Universal Robots PolyScope program: MarinaFerranP3.urp

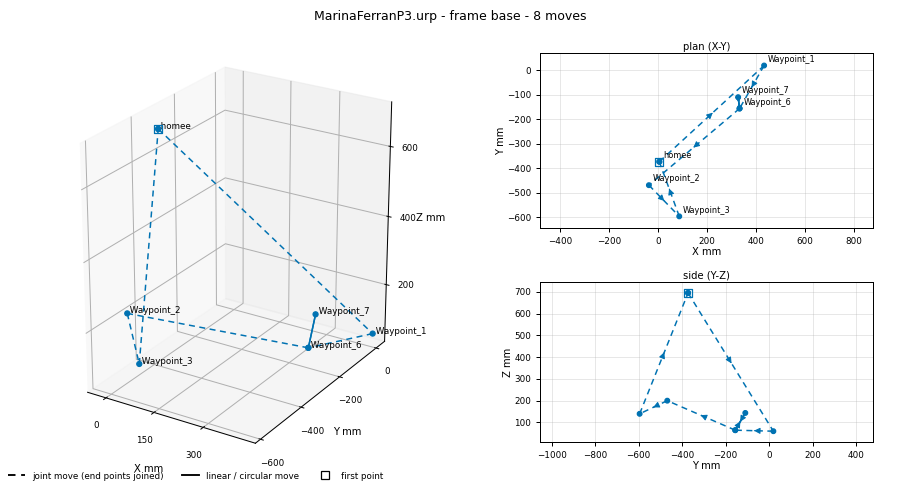
[picture p0: tool path of MarinaFerranP3.urp in frame base, 8 of 8 moves have a stored position in this frame; points joined in program order, loops and branches not executed]
Program MarinaFerranP3 (installation=default directory=/programs createdIn=5.14.5 lastSavedIn=5.14.5 robotSerialNumber=20195300809)
Calibrated DH parameters: a=[-0.000085, -0.20076, -0.212369, 0.000121, -0.000118, 0]; d=[0.15185, -26.306375, 24.753047, 1.684739, 0.085386, 0.092088]; alpha=[1.572149, -0.00522, -0.011864, 1.571339, -1.571085, 0]; deltaTheta=[0, 0.599885, -0.513355, -0.086555, 0.000006, 0]
InitVariablesNode
Robot Program (runOnlyOnce=false)
  URCap Gripper (Robotiq_Grippers, Robotiq Inc.) dataModel(position=0.0, force=100.0, speed=100.0, positionInDouble=0.0, forceInDouble=100.0, speedInDouble=100.0, slaveIds=[9], blocking=true)
  MoveJ speed 60 deg/s, acceleration 80 deg/s^2 (useActiveTCP=true) feature=Base
    Waypoint homee: TCP in base x=5.952 y=-372.701 z=694.671 mm, rx=-0.0179 ry=2.2102 rz=-2.2166 rad; joints [-0.001, -90.001, 0, -89.999, 0.001, -0.002] deg; TCP offset x=0 y=0 z=150 mm, rx=0 ry=0 rz=0 rad
    Waypoint Waypoint_1: TCP in base x=432.947 y=19.396 z=59.118 mm, rx=0.0268 ry=3.127 rz=-0.1601 rad; joints [23.277, -120.171, -75.596, -76.061, 83.68, 114.572] deg; TCP offset x=0 y=0 z=150 mm, rx=0 ry=0 rz=0 rad
    URCap Gripper (Robotiq_Grippers, Robotiq Inc.) dataModel(position=100.0, force=100.0, speed=100.0, positionInDouble=100.0, forceInDouble=100.0, speedInDouble=100.0, slaveIds=[9], blocking=true)
    Waypoint Waypoint_6: TCP in base x=332.939 y=-155.806 z=63.764 mm, rx=-0.1442 ry=3.0939 rz=-0.1586 rad; joints [-0.24, -100.37, -104.415, -62.59, 83.669, 84.337] deg; TCP offset x=0 y=0 z=150 mm, rx=0 ry=0 rz=0 rad
    MoveL speed 250 mm/s, acceleration 1200 mm/s^2 (useActiveTCP=true) feature=Base
      Waypoint Waypoint_7: TCP in base x=327.175 y=-109.602 z=143.022 mm, rx=1.9172 ry=2.2694 rz=-0.0775 rad; joints [10.932, -86.812, -97.987, -81.402, 79.971, 181.23] deg; TCP offset x=0 y=0 z=150 mm, rx=0 ry=0 rz=0 rad
      Waypoint Waypoint_8: TCP in base x=332.951 y=-155.779 z=63.766 mm, rx=-0.1442 ry=3.0939 rz=-0.1585 rad; joints [-0.239, -100.371, -104.413, -62.591, 83.673, 84.338] deg; TCP offset x=0 y=0 z=150 mm, rx=0 ry=0 rz=0 rad
    Waypoint Waypoint_2: TCP in base x=-36.61 y=-468.27 z=199.401 mm, rx=1.7288 ry=1.9459 rz=-0.7398 rad; joints [-70.762, -93.264, -103.578, -35.004, 75.56, 97.405] deg; TCP offset x=0 y=0 z=150 mm, rx=0 ry=0 rz=0 rad
    Force Frame feature=Plane_1; selection=[1, 1, 0, 0, 0, 0]; wrench=[0, 0, 0, 0, 0, 0]; limitsForce=[0.15, 0.15, 0.15, 1.047198, 1.047198, 1.047198]; limitsMotion=[0.1, 0.1, 0.1, 0.349066, 0.349066, 0.349066]
      Waypoint Waypoint_3: TCP in base x=87.13 y=-595.333 z=139.042 mm, rx=1.7042 ry=1.8262 rz=-0.6959 rad; joints [-62.269, -129.159, -73.464, -25.94, 72.716, 107.036] deg
      var_1 :=  (valueSource=Operator valueType=Boolean)
    Force Frame feature=Plane_1; selection=[0, 0, 1, 0, 0, 0]; wrench=[0, 0, -5, 0, 0, 0]; limitsForce=[0.15, 0.15, 0.15, 1.047198, 1.047198, 1.047198]; limitsMotion=[0.1, 0.1, 0.1, 0.349066, 0.349066, 0.349066]
      Wait Sleep waitTime=5
    URCap Gripper (Robotiq_Grippers, Robotiq Inc.) dataModel(position=0.0, force=100.0, speed=100.0, positionInDouble=0.0, forceInDouble=100.0, speedInDouble=100.0, slaveIds=[9], blocking=true)
    Force Frame feature=Plane_1; selection=[0, 0, 1, 0, 0, 0]; wrench=[0, 0, 5, 0, 0, 0]; limitsForce=[0.15, 0.15, 0.15, 1.047198, 1.047198, 1.047198]; limitsMotion=[0.1, 0.1, 0.1, 0.349066, 0.349066, 0.349066]
      Wait Sleep waitTime=3
    MoveJ speed 60 deg/s, acceleration 80 deg/s^2 (useActiveTCP=true) feature=Base
      Waypoint Waypoint_5: TCP in base x=5.911 y=-372.701 z=694.671 mm, rx=-0.0178 ry=2.2102 rz=-2.2165 rad; joints [-0.003, -90, 0.001, -89.999, -0.001, 0] deg
    Popup Message (haltProgram=false message=Se acabo inputType=Text)
